Yaskawa INFORM job: argaz5.JBI

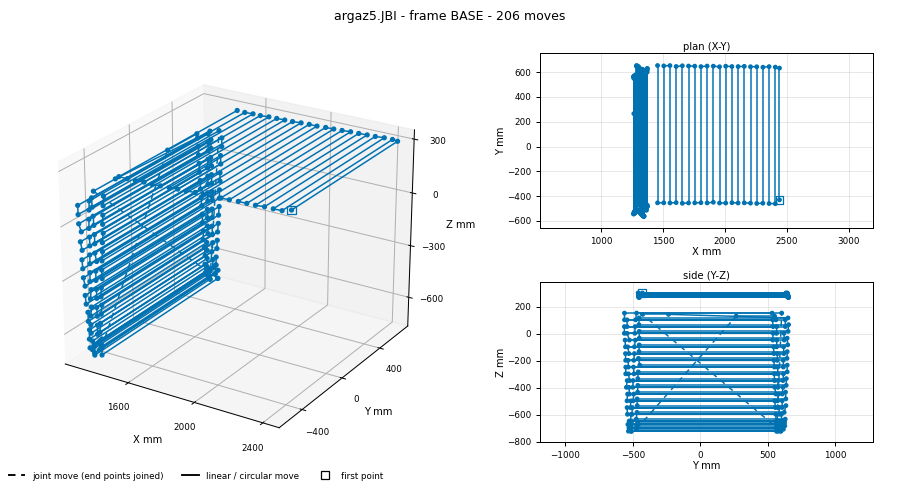
[picture p0: tool path of argaz5.JBI in frame BASE, 206 of 212 moves have a stored position in this frame; points joined in program order, loops and branches not executed]
/JOB
//NAME ARGAZ5
//POS
///NPOS 206,0,206,0,0,0
///TOOL 0
///POSTYPE BASE
///RECTAN
///RCONF 0,0,0,0,0,0,0,0,0,0,0,0,0,0,0,0,0,0,0,0,0,0,0,0
C00000=2438.372582,-429.843151,302.316766,175.000000,5.000000,175.000000
C00001=2438.372582,633.343784,302.316766,175.000000,5.000000,175.000000
C00002=2404.704851,640.901807,302.803619,175.000000,5.000000,175.000000
C00003=2404.704851,-461.113938,302.803619,175.000000,5.000000,175.000000
C00004=2354.704851,-459.538033,300.563623,175.000000,5.000000,175.000000
C00005=2354.704851,645.007128,300.563623,175.000000,5.000000,175.000000
C00006=2304.704851,639.966157,299.253108,175.000000,5.000000,175.000000
C00007=2304.704851,-457.215394,299.253108,175.000000,5.000000,175.000000
C00008=2254.704851,-459.172566,296.365196,175.000000,5.000000,175.000000
C00009=2254.704851,644.031634,296.365196,175.000000,5.000000,175.000000
C00010=2204.704851,644.248715,294.144178,175.000000,5.000000,175.000000
C00011=2204.704851,-456.654141,294.144178,175.000000,5.000000,175.000000
C00012=2154.704851,-454.150829,292.149481,175.000000,5.000000,175.000000
C00013=2154.704851,647.282366,292.149481,175.000000,5.000000,175.000000
C00014=2104.704851,645.426179,290.068247,175.000000,5.000000,175.000000
C00015=2104.704851,-455.328293,290.068247,175.000000,5.000000,175.000000
C00016=2054.704851,-453.054428,287.793100,175.000000,5.000000,175.000000
C00017=2054.704851,645.839734,287.793100,175.000000,5.000000,175.000000
C00018=2004.704851,648.293583,285.625121,175.000000,5.000000,175.000000
C00019=2004.704851,-455.974043,285.625121,175.000000,5.000000,175.000000
C00020=1954.704851,-455.663533,284.513942,175.000000,5.000000,175.000000
C00021=1954.704851,644.044686,284.513942,175.000000,5.000000,175.000000
C00022=1904.704851,648.760722,282.533752,175.000000,5.000000,175.000000
C00023=1904.704851,-449.454029,282.533752,175.000000,5.000000,175.000000
C00024=1854.704851,-454.861154,280.617582,175.000000,5.000000,175.000000
C00025=1854.704851,649.609814,280.617582,175.000000,5.000000,175.000000
C00026=1804.704851,645.165131,279.272701,175.000000,5.000000,175.000000
C00027=1804.704851,-453.058550,279.272701,175.000000,5.000000,175.000000
C00028=1754.704851,-454.350050,276.998525,175.000000,5.000000,175.000000
C00029=1754.704851,648.797818,276.998525,175.000000,5.000000,175.000000
C00030=1704.704851,649.851627,275.425867,175.000000,5.000000,175.000000
C00031=1704.704851,-455.236239,275.425867,175.000000,5.000000,175.000000
C00032=1654.704851,-457.856335,273.661155,175.000000,5.000000,175.000000
C00033=1654.704851,651.982602,273.661155,175.000000,5.000000,175.000000
C00034=1604.704851,646.210696,272.661528,175.000000,5.000000,175.000000
C00035=1604.704851,-452.258232,272.661528,175.000000,5.000000,175.000000
C00036=1554.704851,-455.193647,270.474072,175.000000,5.000000,175.000000
C00037=1554.704851,653.496680,270.474072,175.000000,5.000000,175.000000
C00038=1504.704851,650.879331,269.338933,175.000000,5.000000,175.000000
C00039=1504.704851,-454.045036,269.338933,175.000000,5.000000,175.000000
C00040=1454.676558,-454.040915,269.843337,175.000000,5.000000,175.000000
C00041=1454.676558,653.895121,269.843337,175.000000,5.000000,175.000000
C00042=1347.088440,531.287212,153.366162,175.000000,-89.999999,5.000000
C00043=1347.088440,-562.394236,153.366162,175.000000,-89.999999,5.000000
C00044=1344.164261,-562.287069,103.366162,175.000000,-89.999999,5.000000
C00045=1344.164261,534.938218,103.366162,175.000000,-89.999999,5.000000
C00046=1342.438438,538.625405,53.366162,175.000000,-89.999999,5.000000
C00047=1342.438438,-562.994646,53.366162,175.000000,-89.999999,5.000000
C00048=1340.832322,-563.178754,3.366162,175.000000,-89.999999,5.000000
C00049=1340.832322,538.871340,3.366162,175.000000,-89.999999,5.000000
C00050=1338.825152,536.219643,-46.633838,175.000000,-89.999999,5.000000
C00051=1338.825152,-558.107555,-46.633838,175.000000,-89.999999,5.000000
C00052=1337.044766,-554.870562,-96.633838,175.000000,-89.999999,5.000000
C00053=1337.044766,542.164664,-96.633838,175.000000,-89.999999,5.000000
C00054=1335.183955,545.111757,-146.633838,175.000000,-89.999999,5.000000
C00055=1335.183955,-555.018947,-146.633838,175.000000,-89.999999,5.000000
C00056=1333.293055,-553.493878,-196.633838,175.000000,-89.999999,5.000000
C00057=1333.293055,545.184576,-196.633838,175.000000,-89.999999,5.000000
C00058=1331.807234,548.689487,-246.633838,175.000000,-89.999999,5.000000
C00059=1331.807234,-552.923694,-246.633838,175.000000,-89.999999,5.000000
C00060=1329.870905,-553.256187,-296.633838,175.000000,-89.999999,5.000000
C00061=1329.870905,547.209758,-296.633838,175.000000,-89.999999,5.000000
C00062=1327.995986,549.873820,-346.633838,175.000000,-89.999999,5.000000
C00063=1327.995986,-542.334769,-346.633838,175.000000,-89.999999,5.000000
C00064=1326.213293,-548.248877,-396.633838,175.000000,-89.999999,5.000000
C00065=1326.213293,550.626737,-396.633838,175.000000,-89.999999,5.000000
C00066=1324.396229,560.131627,-446.633838,175.000000,-89.999999,5.000000
C00067=1324.396229,-539.231047,-446.633838,175.000000,-89.999999,5.000000
C00068=1322.129137,-543.451779,-496.633838,175.000000,-89.999999,5.000000
C00069=1322.129137,550.722913,-496.633838,175.000000,-89.999999,5.000000
C00070=1320.170759,556.350555,-546.633838,175.000000,-89.999999,5.000000
C00071=1320.170759,-543.270419,-546.633838,175.000000,-89.999999,5.000000
C00072=1318.250549,-540.170819,-596.633838,175.000000,-89.999999,5.000000
C00073=1318.250549,558.973399,-596.633838,175.000000,-89.999999,5.000000
C00074=1316.642116,560.301995,-646.633838,175.000000,-89.999999,5.000000
C00075=1316.642116,-527.964771,-646.633838,175.000000,-89.999999,5.000000
C00076=1314.806880,-529.352446,-696.633838,175.000000,-89.999999,5.000000
C00077=1314.806880,561.085139,-696.633838,175.000000,-89.999999,5.000000
C00078=1333.412797,565.195956,-671.633838,180.000000,-60.000000,0.000000
C00079=1333.412797,-537.251205,-671.633838,180.000000,-60.000000,0.000000
C00080=1332.156410,-533.079935,-721.633838,180.000000,-60.000000,0.000000
C00081=1332.156410,565.345715,-721.633838,180.000000,-60.000000,0.000000
C00082=1332.156410,565.345715,-721.633838,180.000000,-60.000000,0.000000
C00083=1371.377692,602.641704,153.649998,175.000000,-89.999999,5.000000
C00084=1371.377692,-472.613364,153.649998,175.000000,-89.999999,5.000000
C00085=1372.180185,-480.408458,103.649998,175.000000,-89.999999,5.000000
C00086=1372.180185,629.123405,103.649998,175.000000,-89.999999,5.000000
C00087=1371.089827,629.796808,53.649998,175.000000,-89.999999,5.000000
C00088=1371.089827,-483.667374,53.649998,175.000000,-89.999999,5.000000
C00089=1369.998045,-485.573285,3.649998,175.000000,-89.999999,5.000000
C00090=1369.998045,619.394857,3.649998,175.000000,-89.999999,5.000000
C00091=1369.110863,621.830265,-46.350002,175.000000,-89.999999,5.000000
C00092=1369.110863,-481.873008,-46.350002,175.000000,-89.999999,5.000000
C00093=1367.639331,-488.976108,-96.350002,175.000000,-89.999999,5.000000
C00094=1367.639331,616.630322,-96.350002,175.000000,-89.999999,5.000000
C00095=1366.582076,618.500428,-146.350002,175.000000,-89.999999,5.000000
C00096=1366.582076,-488.746131,-146.350002,175.000000,-89.999999,5.000000
C00097=1365.085299,-493.213455,-196.350002,175.000000,-89.999999,5.000000
C00098=1365.085299,614.650047,-196.350002,175.000000,-89.999999,5.000000
C00099=1363.658730,614.990191,-246.350002,175.000000,-89.999999,5.000000
C00100=1363.658730,-495.754211,-246.350002,175.000000,-89.999999,5.000000
C00101=1361.864342,-491.909338,-296.350002,175.000000,-89.999999,5.000000
C00102=1361.864342,615.571329,-296.350002,175.000000,-89.999999,5.000000
C00103=1360.073877,611.872429,-346.350002,175.000000,-89.999999,5.000000
C00104=1360.073877,-498.655768,-346.350002,175.000000,-89.999999,5.000000
C00105=1358.161888,-500.748966,-396.350002,175.000000,-89.999999,5.000000
C00106=1358.161888,611.928890,-396.350002,175.000000,-89.999999,5.000000
C00107=1356.405837,607.009877,-446.350002,175.000000,-89.999999,5.000000
C00108=1356.405837,-493.709213,-446.350002,175.000000,-89.999999,5.000000
C00109=1354.608405,-498.341789,-496.350002,175.000000,-89.999999,5.000000
C00110=1354.608405,606.376409,-496.350002,175.000000,-89.999999,5.000000
C00111=1352.468508,605.807665,-546.350002,175.000000,-89.999999,5.000000
C00112=1352.468508,-503.981028,-546.350002,175.000000,-89.999999,5.000000
C00113=1350.405576,-507.600056,-596.350002,175.000000,-89.999999,5.000000
C00114=1350.405576,600.519588,-596.350002,175.000000,-89.999999,5.000000
C00115=1348.479511,602.258869,-646.350002,175.000000,-89.999999,5.000000
C00116=1348.479511,-507.412770,-646.350002,175.000000,-89.999999,5.000000
C00117=1346.462576,-509.588593,-696.350002,175.000000,-89.999999,5.000000
C00118=1346.462576,597.739216,-696.350002,175.000000,-89.999999,5.000000
C00119=1364.869259,596.218205,-671.350002,180.000000,-60.000000,0.000000
C00120=1364.869259,-512.867477,-671.350002,180.000000,-60.000000,0.000000
C00121=1363.104675,-512.908790,-721.350002,180.000000,-60.000000,0.000000
C00122=1363.104675,596.344210,-721.350002,180.000000,-60.000000,0.000000
C00123=1363.104675,596.344210,-721.350002,180.000000,-60.000000,0.000000
C00124=1277.888245,-429.618923,144.199188,175.000000,-89.999999,5.000000
C00125=1277.888245,-236.558107,144.199188,175.000000,-89.999999,5.000000
C00126=1283.410944,649.398505,117.816493,175.000000,-89.999999,5.000000
C00127=1283.410944,-454.812790,117.816493,175.000000,-89.999999,5.000000
C00128=1286.253415,-455.480523,67.816493,175.000000,-89.999999,5.000000
C00129=1286.253415,653.737395,67.816493,175.000000,-89.999999,5.000000
C00130=1288.733474,650.101960,17.816493,175.000000,-89.999999,5.000000
C00131=1288.733474,-453.231390,17.816493,175.000000,-89.999999,5.000000
C00132=1291.050491,-452.345201,-32.183507,175.000000,-89.999999,5.000000
C00133=1291.050491,643.233653,-32.183507,175.000000,-89.999999,5.000000
C00134=1293.592039,647.319739,-82.183507,175.000000,-89.999999,5.000000
C00135=1293.592039,-453.386645,-82.183507,175.000000,-89.999999,5.000000
C00136=1295.614737,-454.881487,-132.183507,175.000000,-89.999999,5.000000
C00137=1295.614737,643.520806,-132.183507,175.000000,-89.999999,5.000000
C00138=1297.247512,642.008789,-182.183507,175.000000,-89.999999,5.000000
C00139=1297.247512,-459.228621,-182.183507,175.000000,-89.999999,5.000000
C00140=1299.433219,-449.216748,-232.183507,175.000000,-89.999999,5.000000
C00141=1299.433219,643.471344,-232.183507,175.000000,-89.999999,5.000000
C00142=1300.418371,643.420508,-282.183507,175.000000,-89.999999,5.000000
C00143=1300.418371,-460.256325,-282.183507,175.000000,-89.999999,5.000000
C00144=1302.234326,-463.734445,-332.183507,175.000000,-89.999999,5.000000
C00145=1302.234326,636.925912,-332.183507,175.000000,-89.999999,5.000000
C00146=1303.707506,635.868668,-382.183507,175.000000,-89.999999,5.000000
C00147=1303.707506,-463.869777,-382.183507,175.000000,-89.999999,5.000000
C00148=1305.086846,-465.019762,-432.183507,175.000000,-89.999999,5.000000
C00149=1305.086846,630.756939,-432.183507,175.000000,-89.999999,5.000000
C00150=1306.071877,633.429245,-482.183507,175.000000,-89.999999,5.000000
C00151=1306.071877,-468.802208,-482.183507,175.000000,-89.999999,5.000000
C00152=1307.412042,-468.117988,-532.183507,175.000000,-89.999999,5.000000
C00153=1307.412042,633.875774,-532.183507,175.000000,-89.999999,5.000000
C00154=1308.466459,621.089237,-582.183507,175.000000,-89.999999,5.000000
C00155=1308.466459,-469.996158,-582.183507,175.000000,-89.999999,5.000000
C00156=1310.304432,-475.204750,-632.183507,175.000000,-89.999999,5.000000
C00157=1310.304432,628.888386,-632.183507,175.000000,-89.999999,5.000000
C00158=1311.312316,625.813517,-682.183507,175.000000,-89.999999,5.000000
C00159=1311.312316,-473.494887,-682.183507,175.000000,-89.999999,5.000000
C00160=1332.658786,-465.818706,-657.183507,180.000000,-60.000000,0.000000
C00161=1332.658786,624.168915,-657.183507,180.000000,-60.000000,0.000000
C00162=1333.118383,615.110554,-707.183507,180.000000,-60.000000,0.000000
C00163=1333.118383,-474.618080,-707.183507,180.000000,-60.000000,0.000000
C00164=1333.118383,-474.618080,-707.183507,180.000000,-60.000000,0.000000
C00165=1263.288256,265.502746,131.277012,175.000000,-89.999999,5.000000
C00166=1263.288256,550.035994,131.277012,175.000000,-89.999999,5.000000
C00167=1260.890439,559.755591,103.296988,175.000000,-89.999999,5.000000
C00168=1260.890439,-543.266015,103.296988,175.000000,-89.999999,5.000000
C00169=1261.533657,-543.209554,53.296988,175.000000,-89.999999,5.000000
C00170=1261.533657,565.502244,53.296988,175.000000,-89.999999,5.000000
C00171=1263.366070,564.257342,3.296988,175.000000,-89.999999,5.000000
C00172=1263.366070,-543.096632,3.296988,175.000000,-89.999999,5.000000
C00173=1265.404717,-525.948939,-46.703012,175.000000,-89.999999,5.000000
C00174=1265.404717,566.502021,-46.703012,175.000000,-89.999999,5.000000
C00175=1267.028835,564.815069,-96.703012,175.000000,-89.999999,5.000000
C00176=1267.028835,-538.386938,-96.703012,175.000000,-89.999999,5.000000
C00177=1269.183844,-528.977189,-146.703012,175.000000,-89.999999,5.000000
C00178=1269.183844,570.662251,-146.703012,175.000000,-89.999999,5.000000
C00179=1270.966410,569.787790,-196.703012,175.000000,-89.999999,5.000000
C00180=1270.966410,-535.503283,-196.703012,175.000000,-89.999999,5.000000
C00181=1272.925389,-533.396314,-246.703012,175.000000,-89.999999,5.000000
C00182=1272.925389,572.645280,-246.703012,175.000000,-89.999999,5.000000
C00183=1275.047149,573.565873,-296.703012,175.000000,-89.999999,5.000000
C00184=1275.047149,-533.499597,-296.703012,175.000000,-89.999999,5.000000
C00185=1277.369843,-524.427239,-346.703012,175.000000,-89.999999,5.000000
C00186=1277.369843,576.345557,-346.703012,175.000000,-89.999999,5.000000
C00187=1279.521115,573.757979,-396.703012,175.000000,-89.999999,5.000000
C00188=1279.521115,-528.930368,-396.703012,175.000000,-89.999999,5.000000
C00189=1281.635581,-525.764407,-446.703012,175.000000,-89.999999,5.000000
C00190=1281.635581,579.175964,-446.703012,175.000000,-89.999999,5.000000
C00191=1283.849911,571.736391,-496.703012,175.000000,-89.999999,5.000000
C00192=1283.849911,-515.793718,-496.703012,175.000000,-89.999999,5.000000
C00193=1285.977049,-517.912163,-546.703012,175.000000,-89.999999,5.000000
C00194=1285.977049,582.744957,-546.703012,175.000000,-89.999999,5.000000
C00195=1288.303918,585.349060,-596.703012,175.000000,-89.999999,5.000000
C00196=1288.303918,-512.618577,-596.703012,175.000000,-89.999999,5.000000
C00197=1290.270344,-519.107488,-646.703012,175.000000,-89.999999,5.000000
C00198=1290.270344,579.567979,-646.703012,175.000000,-89.999999,5.000000
C00199=1292.656383,581.655668,-696.703012,175.000000,-89.999999,5.000000
C00200=1292.656383,-518.761835,-696.703012,175.000000,-89.999999,5.000000
C00201=1314.870088,-511.376429,-671.703012,180.000000,-60.000000,0.000000
C00202=1314.870088,581.349951,-671.703012,180.000000,-60.000000,0.000000
C00203=1317.105759,581.261816,-721.703012,180.000000,-60.000000,0.000000
C00204=1317.105759,-511.969961,-721.703012,180.000000,-60.000000,0.000000
C00205=1317.105759,-511.969961,-721.703012,180.000000,-60.000000,0.000000
///POSTYPE PULSE
///PULSE
EC00000=0
EC00001=0
EC00002=0
EC00003=0
EC00004=0
EC00005=0
EC00006=0
EC00007=0
EC00008=0
EC00009=0
EC00010=0
EC00011=0
EC00012=0
EC00013=0
EC00014=0
EC00015=0
EC00016=0
EC00017=0
EC00018=0
EC00019=0
EC00020=0
EC00021=0
EC00022=0
EC00023=0
EC00024=0
EC00025=0
EC00026=0
EC00027=0
EC00028=0
EC00029=0
EC00030=0
EC00031=0
EC00032=0
EC00033=0
EC00034=0
EC00035=0
EC00036=0
EC00037=0
EC00038=0
EC00039=0
EC00040=0
EC00041=0
EC00042=0
EC00043=0
EC00044=0
EC00045=0
EC00046=0
EC00047=0
EC00048=0
EC00049=0
EC00050=0
EC00051=0
EC00052=0
EC00053=0
EC00054=0
EC00055=0
EC00056=0
EC00057=0
EC00058=0
EC00059=0
EC00060=0
EC00061=0
EC00062=0
EC00063=0
EC00064=0
EC00065=0
EC00066=0
EC00067=0
EC00068=0
EC00069=0
EC00070=0
EC00071=0
EC00072=0
EC00073=0
EC00074=0
EC00075=0
EC00076=0
EC00077=0
EC00078=0
EC00079=0
EC00080=0
EC00081=0
EC00082=92160
EC00083=92160
EC00084=92160
EC00085=92160
EC00086=92160
EC00087=92160
EC00088=92160
EC00089=92160
EC00090=92160
EC00091=92160
EC00092=92160
EC00093=92160
EC00094=92160
EC00095=92160
EC00096=92160
EC00097=92160
EC00098=92160
EC00099=92160
EC00100=92160
EC00101=92160
EC00102=92160
EC00103=92160
EC00104=92160
EC00105=92160
EC00106=92160
EC00107=92160
EC00108=92160
EC00109=92160
EC00110=92160
EC00111=92160
EC00112=92160
EC00113=92160
EC00114=92160
EC00115=92160
EC00116=92160
EC00117=92160
EC00118=92160
EC00119=92160
EC00120=92160
EC00121=92160
EC00122=92160
EC00123=184320
EC00124=184320
EC00125=184320
EC00126=184320
EC00127=184320
EC00128=184320
EC00129=184320
EC00130=184320
EC00131=184320
EC00132=184320
EC00133=184320
EC00134=184320
EC00135=184320
EC00136=184320
EC00137=184320
EC00138=184320
EC00139=184320
EC00140=184320
EC00141=184320
EC00142=184320
EC00143=184320
EC00144=184320
EC00145=184320
EC00146=184320
EC00147=184320
EC00148=184320
EC00149=184320
EC00150=184320
EC00151=184320
EC00152=184320
EC00153=184320
EC00154=184320
EC00155=184320
EC00156=184320
EC00157=184320
EC00158=184320
EC00159=184320
EC00160=184320
EC00161=184320
EC00162=184320
EC00163=184320
EC00164=276480
EC00165=276480
EC00166=276480
EC00167=276480
EC00168=276480
EC00169=276480
EC00170=276480
EC00171=276480
EC00172=276480
EC00173=276480
EC00174=276480
EC00175=276480
EC00176=276480
EC00177=276480
EC00178=276480
EC00179=276480
EC00180=276480
EC00181=276480
EC00182=276480
EC00183=276480
EC00184=276480
EC00185=276480
EC00186=276480
EC00187=276480
EC00188=276480
EC00189=276480
EC00190=276480
EC00191=276480
EC00192=276480
EC00193=276480
EC00194=276480
EC00195=276480
EC00196=276480
EC00197=276480
EC00198=276480
EC00199=276480
EC00200=276480
EC00201=276480
EC00202=276480
EC00203=276480
EC00204=276480
EC00205=368640
//INST
///DATE 2023/01/29 16:16
///ATTR SC,RW,RJ
////FRAME BASE
///GROUP1 RB1,ST1
NOP
MOVJ P009 EX000 VJ=15.00
MOVJ C00000 EC00000 VJ=15.0
CALL JOB:SPYON
MOVL C00001 EC00001 V=150.0
MOVL C00002 EC00002 V=150.0
MOVL C00003 EC00003 V=150.0
MOVL C00004 EC00004 V=150.0
MOVL C00005 EC00005 V=150.0
MOVL C00006 EC00006 V=150.0
MOVL C00007 EC00007 V=150.0
MOVL C00008 EC00008 V=150.0
MOVL C00009 EC00009 V=150.0
MOVL C00010 EC00010 V=150.0
MOVL C00011 EC00011 V=150.0
MOVL C00012 EC00012 V=150.0
MOVL C00013 EC00013 V=150.0
MOVL C00014 EC00014 V=150.0
MOVL C00015 EC00015 V=150.0
MOVL C00016 EC00016 V=150.0
MOVL C00017 EC00017 V=150.0
MOVL C00018 EC00018 V=150.0
MOVL C00019 EC00019 V=150.0
MOVL C00020 EC00020 V=150.0
MOVL C00021 EC00021 V=150.0
MOVL C00022 EC00022 V=150.0
MOVL C00023 EC00023 V=150.0
MOVL C00024 EC00024 V=150.0
MOVL C00025 EC00025 V=150.0
MOVL C00026 EC00026 V=150.0
MOVL C00027 EC00027 V=150.0
MOVL C00028 EC00028 V=150.0
MOVL C00029 EC00029 V=150.0
MOVL C00030 EC00030 V=150.0
MOVL C00031 EC00031 V=150.0
MOVL C00032 EC00032 V=150.0
MOVL C00033 EC00033 V=150.0
MOVL C00034 EC00034 V=150.0
MOVL C00035 EC00035 V=150.0
MOVL C00036 EC00036 V=150.0
MOVL C00037 EC00037 V=150.0
MOVL C00038 EC00038 V=150.0
MOVL C00039 EC00039 V=150.0
MOVL C00040 EC00040 V=150.0
MOVL C00041 EC00041 V=150.0
CALL JOB:SPYOF
MOVJ P009 VJ=15.00
MOVJ C00042 EC00042 VJ=15.0
CALL JOB:SPYON
MOVL C00043 EC00043 V=150.0
MOVL C00044 EC00044 V=150.0
MOVL C00045 EC00045 V=150.0
MOVL C00046 EC00046 V=150.0
MOVL C00047 EC00047 V=150.0
MOVL C00048 EC00048 V=150.0
MOVL C00049 EC00049 V=150.0
MOVL C00050 EC00050 V=150.0
MOVL C00051 EC00051 V=150.0
MOVL C00052 EC00052 V=150.0
MOVL C00053 EC00053 V=150.0
MOVL C00054 EC00054 V=150.0
MOVL C00055 EC00055 V=150.0
MOVL C00056 EC00056 V=150.0
MOVL C00057 EC00057 V=150.0
MOVL C00058 EC00058 V=150.0
MOVL C00059 EC00059 V=150.0
MOVL C00060 EC00060 V=150.0
MOVL C00061 EC00061 V=150.0
MOVL C00062 EC00062 V=150.0
MOVL C00063 EC00063 V=150.0
MOVL C00064 EC00064 V=150.0
MOVL C00065 EC00065 V=150.0
MOVL C00066 EC00066 V=150.0
MOVL C00067 EC00067 V=150.0
MOVL C00068 EC00068 V=150.0
MOVL C00069 EC00069 V=150.0
MOVL C00070 EC00070 V=150.0
MOVL C00071 EC00071 V=150.0
MOVL C00072 EC00072 V=150.0
MOVL C00073 EC00073 V=150.0
MOVL C00074 EC00074 V=150.0
MOVL C00075 EC00075 V=150.0
MOVL C00076 EC00076 V=150.0
MOVL C00077 EC00077 V=150.0
MOVL C00078 EC00078 V=150.0
MOVL C00079 EC00079 V=150.0
MOVL C00080 EC00080 V=150.0
MOVL C00081 EC00081 V=150.0
CALL JOB:SPYOF
MOVJ P009 VJ=15.00
MOVL C00082 EC00082 V=150.0
MOVJ C00083 EC00083 VJ=15.0
CALL JOB:SPYON
MOVL C00084 EC00084 V=150.0
MOVL C00085 EC00085 V=150.0
MOVL C00086 EC00086 V=150.0
MOVL C00087 EC00087 V=150.0
MOVL C00088 EC00088 V=150.0
MOVL C00089 EC00089 V=150.0
MOVL C00090 EC00090 V=150.0
MOVL C00091 EC00091 V=150.0
MOVL C00092 EC00092 V=150.0
MOVL C00093 EC00093 V=150.0
MOVL C00094 EC00094 V=150.0
MOVL C00095 EC00095 V=150.0
MOVL C00096 EC00096 V=150.0
MOVL C00097 EC00097 V=150.0
MOVL C00098 EC00098 V=150.0
MOVL C00099 EC00099 V=150.0
MOVL C00100 EC00100 V=150.0
MOVL C00101 EC00101 V=150.0
MOVL C00102 EC00102 V=150.0
MOVL C00103 EC00103 V=150.0
MOVL C00104 EC00104 V=150.0
MOVL C00105 EC00105 V=150.0
MOVL C00106 EC00106 V=150.0
MOVL C00107 EC00107 V=150.0
MOVL C00108 EC00108 V=150.0
MOVL C00109 EC00109 V=150.0
MOVL C00110 EC00110 V=150.0
MOVL C00111 EC00111 V=150.0
MOVL C00112 EC00112 V=150.0
MOVL C00113 EC00113 V=150.0
MOVL C00114 EC00114 V=150.0
MOVL C00115 EC00115 V=150.0
MOVL C00116 EC00116 V=150.0
MOVL C00117 EC00117 V=150.0
MOVL C00118 EC00118 V=150.0
MOVL C00119 EC00119 V=150.0
MOVL C00120 EC00120 V=150.0
MOVL C00121 EC00121 V=150.0
MOVL C00122 EC00122 V=150.0
CALL JOB:SPYOF
MOVJ P009 VJ=15.00
MOVL C00123 EC00123 V=150.0
MOVJ C00124 EC00124 VJ=15.0
CALL JOB:SPYON
MOVL C00125 EC00125 V=150.0
MOVL C00126 EC00126 V=150.0
MOVL C00127 EC00127 V=150.0
MOVL C00128 EC00128 V=150.0
MOVL C00129 EC00129 V=150.0
MOVL C00130 EC00130 V=150.0
MOVL C00131 EC00131 V=150.0
MOVL C00132 EC00132 V=150.0
MOVL C00133 EC00133 V=150.0
MOVL C00134 EC00134 V=150.0
MOVL C00135 EC00135 V=150.0
MOVL C00136 EC00136 V=150.0
MOVL C00137 EC00137 V=150.0
MOVL C00138 EC00138 V=150.0
MOVL C00139 EC00139 V=150.0
MOVL C00140 EC00140 V=150.0
MOVL C00141 EC00141 V=150.0
MOVL C00142 EC00142 V=150.0
MOVL C00143 EC00143 V=150.0
MOVL C00144 EC00144 V=150.0
MOVL C00145 EC00145 V=150.0
MOVL C00146 EC00146 V=150.0
MOVL C00147 EC00147 V=150.0
MOVL C00148 EC00148 V=150.0
MOVL C00149 EC00149 V=150.0
MOVL C00150 EC00150 V=150.0
MOVL C00151 EC00151 V=150.0
MOVL C00152 EC00152 V=150.0
MOVL C00153 EC00153 V=150.0
MOVL C00154 EC00154 V=150.0
MOVL C00155 EC00155 V=150.0
MOVL C00156 EC00156 V=150.0
MOVL C00157 EC00157 V=150.0
MOVL C00158 EC00158 V=150.0
MOVL C00159 EC00159 V=150.0
MOVL C00160 EC00160 V=150.0
MOVL C00161 EC00161 V=150.0
MOVL C00162 EC00162 V=150.0
MOVL C00163 EC00163 V=150.0
CALL JOB:SPYOF
MOVJ P009 VJ=15.00
MOVL C00164 EC00164 V=150.0
MOVJ C00165 EC00165 VJ=15.0
CALL JOB:SPYON
MOVL C00166 EC00166 V=150.0
MOVL C00167 EC00167 V=150.0
MOVL C00168 EC00168 V=150.0
MOVL C00169 EC00169 V=150.0
MOVL C00170 EC00170 V=150.0
MOVL C00171 EC00171 V=150.0
MOVL C00172 EC00172 V=150.0
MOVL C00173 EC00173 V=150.0
MOVL C00174 EC00174 V=150.0
MOVL C00175 EC00175 V=150.0
MOVL C00176 EC00176 V=150.0
MOVL C00177 EC00177 V=150.0
MOVL C00178 EC00178 V=150.0
MOVL C00179 EC00179 V=150.0
MOVL C00180 EC00180 V=150.0
MOVL C00181 EC00181 V=150.0
MOVL C00182 EC00182 V=150.0
MOVL C00183 EC00183 V=150.0
MOVL C00184 EC00184 V=150.0
MOVL C00185 EC00185 V=150.0
MOVL C00186 EC00186 V=150.0
MOVL C00187 EC00187 V=150.0
MOVL C00188 EC00188 V=150.0
MOVL C00189 EC00189 V=150.0
MOVL C00190 EC00190 V=150.0
MOVL C00191 EC00191 V=150.0
MOVL C00192 EC00192 V=150.0
MOVL C00193 EC00193 V=150.0
MOVL C00194 EC00194 V=150.0
MOVL C00195 EC00195 V=150.0
MOVL C00196 EC00196 V=150.0
MOVL C00197 EC00197 V=150.0
MOVL C00198 EC00198 V=150.0
MOVL C00199 EC00199 V=150.0
MOVL C00200 EC00200 V=150.0
MOVL C00201 EC00201 V=150.0
MOVL C00202 EC00202 V=150.0
MOVL C00203 EC00203 V=150.0
MOVL C00204 EC00204 V=150.0
CALL JOB:SPYOF
MOVJ P009 VJ=15.00
MOVL C00205 EC00205 V=150.0
END
